// TwinCAT 3 PLC project Draairichting_FD
// ProgramVersion: 3.1.4024.0
// libraries:
//   Tc2_Standard, * (Beckhoff Automation GmbH)
//   Tc2_System, * (Beckhoff Automation GmbH)
//   Tc3_Module, * (Beckhoff Automation GmbH)
// project tree:
//   / PlcTask.TcTTO
//   POUs/ MAIN.TcPOU
// (motion and I/O tree: see PLC project trappenhuis_extraverlenging)
// real-time tasks:
//   TASK PlcTask: cycle T#10ms, priority 20, ADS port 350
//   TASK PlcTask1: cycle T#10ms, priority 21, ADS port 351
//   TASK PlcTask2: cycle T#10ms, priority 22, ADS port 352
//   TASK PlcTask3: cycle T#10ms, priority 23, ADS port 353
//   TASK PlcTask4: cycle T#10ms, priority 24, ADS port 354
//   TASK PlcTask5: cycle T#10ms, priority 25, ADS port 355
//   TASK PlcTask6: cycle T#10ms, priority 26, ADS port 356
//   TASK PlcTask7: cycle T#10ms, priority 27, ADS port 357
//   TASK PlcTask8: cycle T#10ms, priority 28, ADS port 358
//   TASK PlcTask9: cycle T#10ms, priority 29, ADS port 359
//   TASK PlcTask10: cycle T#10ms, priority 30, ADS port 360

CONFIGURATION Draairichting_FD
    RESOURCE PLC ON TwinCAT3
        TASK PlcTask(INTERVAL := T#10ms, PRIORITY := 27);
        PROGRAM MAIN WITH PlcTask : MAIN;
    END_RESOURCE
END_CONFIGURATION

// ---- POUs/MAIN.TcPOU
PROGRAM MAIN
VAR
    sensorA, sensorB, motorLinksDraaiend, motorRechtsDraaiend, alarm: BOOL;
    fbFlankSensorA, fbFlankSensorB: R_TRIG; // Rising edge detection for sensors
END_VAR

(*
Draairichting van een motor (2 regel code)

Op de as van een motor worden twee sensoren gemonteerd bv reflex fotocellen.
Bepaal de draairichting met flankdetectie.


Uitbreiding: Om een verplaatsbare pomp niet te beschadigen mag een elektrische motor enkel links draaien. 
Daarom wordt de draairichting gedetecteerd door middel van vorige oefening. 
Wanneer de motor links aanloopt is er normale werking.
Als de motor rechts aanloopt zal hij onmiddellijk stilvallen en een rood alarmlicht zal branden.
*)

fbFlankSensorA(CLK:=sensorA); fbFlankSensorB(CLK:=sensorB);
motorLinksDraaiend := fbFlankSensorA.Q AND NOT sensorB; 
motorRechtsDraaiend := fbFlankSensorB.Q AND NOT sensorA;



// Uitbreiding
alarm := NOT motorLinksDraaiend;

END_PROGRAM
